// TIA Portal V21 export
// export: Created 2026-08-04T02:36:01.2839504Z, ExportSetting WithDefaults, DisplayName Totally Integrated Automation Portal, DisplayVersion V21, DisplayName STEP 7 Professional, DisplayVersion V21, DisplayName STEP 7 Safety, DisplayVersion V21, DisplayName Tech WebApplication, DisplayVersion V21, DisplayName WinCC Basic/Comfort/Advanced, DisplayVersion V21
FUNCTION_BLOCK "LAD_StarDelta"   // FB3, LAD
TITLE = LAD_StarDelta
{ S7_Optimized_Access := 'TRUE' }
NAME : StarDelta
VERSION : 0.1
// 星三角启动：5秒星形启动后自动切换三角形，星角互锁，停止时全复位
// stored: AutoNumber true, IsIECCheckEnabled true, IsRetainMemResEnabled false, MemoryReserve 100, SetENOAutomatically false, UDAEnableTagReadback false
   VAR_INPUT
      Start : Bool;
      Stop : Bool;
   END_VAR
   VAR_OUTPUT
      MainContactor : Bool;
      StarContactor : Bool;
      DeltaContactor : Bool;
   END_VAR
   VAR
      "Timer" : TON_TIME;
   END_VAR
   VAR_TEMP
      SwitchDone : Bool;
   END_VAR
BEGIN

REGION Network 1: Network 1: 启动停止自锁
   // 启动/停止/自锁控制 K1
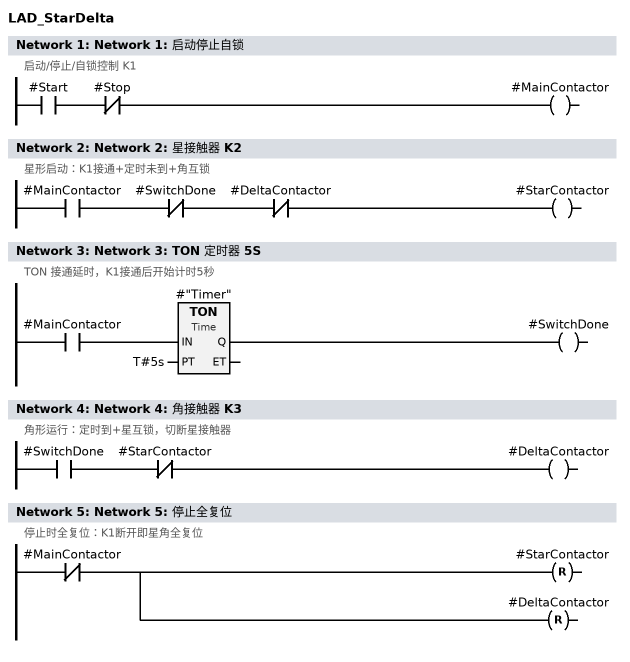
   RUNG wire#powerrail
      Contact( #Start )
      I_Contact( #Stop )
      Coil( #MainContactor )
   END_RUNG
   // the same network as SCL:
   #MainContactor := #Start AND NOT #Stop;
END_REGION

REGION Network 2: Network 2: 星接触器 K2
   // 星形启动：K1接通+定时未到+角互锁
   RUNG wire#powerrail
      Contact( #MainContactor )
      I_Contact( #SwitchDone )
      I_Contact( #DeltaContactor )
      Coil( #StarContactor )
   END_RUNG
   // the same network as SCL:
   #StarContactor := #MainContactor AND NOT #SwitchDone AND NOT #DeltaContactor;
END_REGION

REGION Network 3: Network 3: TON 定时器 5S
   // TON 接通延时，K1接通后开始计时5秒
   RUNG wire#powerrail
      Contact( #MainContactor )
      { S7_Templates := "time_type := Time" } #"Timer".TON(pt := T#5s, et =>)
      Coil( #SwitchDone )
   END_RUNG
   // the same network as SCL:
   #"Timer"(IN := #MainContactor, PT := T#5s);   // TON
   #SwitchDone := #"Timer".Q;
END_REGION

REGION Network 4: Network 4: 角接触器 K3
   // 角形运行：定时到+星互锁，切断星接触器
   RUNG wire#powerrail
      Contact( #SwitchDone )
      I_Contact( #StarContactor )
      Coil( #DeltaContactor )
   END_RUNG
   // the same network as SCL:
   #DeltaContactor := #SwitchDone AND NOT #StarContactor;
END_REGION

REGION Network 5: Network 5: 停止全复位
   // 停止时全复位：K1断开即星角全复位
   RUNG wire#powerrail
      I_Contact( #MainContactor )
      wire#w1
      R_Coil( #StarContactor )
   END_RUNG
   RUNG wire#w1
      R_Coil( #DeltaContactor )
   END_RUNG
   // the same network as SCL:
   IF NOT #MainContactor THEN
       #StarContactor := FALSE;
       #DeltaContactor := FALSE;
   END_IF;
END_REGION
END_FUNCTION_BLOCK
